FUNCTION_BLOCK FemtoCtrl
VAR
	nGainBits AT %Q*: WORD; // assign multiple output bits with correct offset
	bGainMode AT %Q*: BOOL; // TRUE: high gain, FALSE: low gain
	bOverload AT %I*: BOOL;
END_VAR

METHOD GetGain : WORD
VAR_INPUT
END_VAR
GetGain := nGainBits;
END_METHOD

METHOD GetGainMode : BOOL
VAR_INPUT
END_VAR
GetGainMode := bGainMode;
END_METHOD

METHOD GetOverload : BOOL
VAR_INPUT
END_VAR
GetOverload := bOverload;
END_METHOD

METHOD SetGain
VAR_INPUT
	nGain: WORD;
END_VAR
nGainBits := nGain;
END_METHOD

METHOD SetGainMode
VAR_INPUT
	bGainHigh: BOOL;
END_VAR
bGainMode := bGainHigh;
END_METHOD

END_FUNCTION_BLOCK

(* stored: Version 1.1.0.1, ProductVersion 3.1.4024.12
   POU FemtoCtrl: Id {47c97f27-2b8d-47a2-b595-5f9aae5bbedf}, SpecialFunc None
   Method GetGain: Id {081894b6-9955-4205-835f-df5f0efa6ce1}
   Method GetGainMode: Id {536b6c70-298e-4105-ad43-e357434982b5}
   Method GetOverload: Id {54060538-661f-41af-863c-eab994073f8f}
   Method SetGain: Id {86ce544b-1d96-4e41-bd10-3c48c4575352}
   Method SetGainMode: Id {98a5761d-a6dd-4fc6-aa41-ca05541aa048} *)
